FUNCTION RAD_TO_HOUR : LREAL
VAR_INPUT
    rad : LREAL;
END_VAR
VAR
END_VAR

RAD_TO_HOUR := rad * 12.0 / PI;

END_FUNCTION

(* stored: Version 1.1.0.1, ProductVersion 3.1.4018.5
   POU RAD_TO_HOUR: Id {4c241ac3-9c1a-485d-b8de-b30ff65ac587}, SpecialFunc None *)
